// TIA Portal V20 export
TYPE "LBP_typeModularMcpUniversalOutput"
TITLE = Modular MCP image / Image MCP modulaire
// Output image of universal keypad for modular MCP / Image des sorties du pupitre universel pour MCP modulaires
   STRUCT
      led0 : Bool;   // output image n+0 bit 0 / Image des sorties n+0 bit 0
      led1 : Bool;   // output image n+0 bit 1 / Image des sorties n+0 bit 1
      led2 : Bool;   // output image n+0 bit 2 / Image des sorties n+0 bit 2
      led3 : Bool;   // output image n+0 bit 3 / Image des sorties n+0 bit 3
      led4 : Bool;   // output image n+0 bit 4 / Image des sorties n+0 bit 4
      led5 : Bool;   // output image n+0 bit 5 / Image des sorties n+0 bit 5
      led6 : Bool;   // output image n+0 bit 6 / Image des sorties n+0 bit 6
      led7 : Bool;   // output image n+0 bit 7 / Image des sorties n+0 bit 7
      led8 : Bool;   // output image n+1 bit 0 / Image des sorties n+1 bit 0
      led9 : Bool;   // output image n+1 bit 1 / Image des sorties n+1 bit 1
      led10 : Bool;   // output image n+1 bit 2 / Image des sorties n+1 bit 2
      led11 : Bool;   // output image n+1 bit 3 / Image des sorties n+1 bit 3
      led12 : Bool;   // output image n+1 bit 4 / Image des sorties n+1 bit 4
      led13 : Bool;   // output image n+1 bit 5 / Image des sorties n+1 bit 5
      led14 : Bool;   // output image n+1 bit 6 / Image des sorties n+1 bit 6
      reserved17 : Bool;
      led16 : Bool;   // output image n+2 bit 0 / Image des sorties n+2 bit 0
      led17 : Bool;   // output image n+2 bit 1 / Image des sorties n+2 bit 1
      led18 : Bool;   // output image n+2 bit 2 / Image des sorties n+2 bit 2
      reserved23 : Bool;
      reserved24 : Bool;
      reserved25 : Bool;
      reserved26 : Bool;
      reserved27 : Bool;
      led24 : Bool;   // output image n+3 bit 0 / Image des sorties n+3 bit 0
      led25 : Bool;   // output image n+3 bit 1 / Image des sorties n+3 bit 1
      led26 : Bool;   // output image n+3 bit 2 / Image des sorties n+3 bit 2
      reserved33 : Bool;
      reserved34 : Bool;
      reserved35 : Bool;
      reserved36 : Bool;
      reserved37 : Bool;
   END_STRUCT;
END_TYPE
